// Represents the days of the week.
{attribute 'qualified_only'}
{attribute 'to_string'}
TYPE E_DayOfWeek :
(
	_ := 0, // Uninitialised or default value, representing an undefined day.
	Monday,
	Tuesday,
	Wednesday,
	Thursday,
	Friday,
	Saturday,
	Sunday
) UINT;
END_TYPE

(* stored: Version 1.1.0.1
   EnumerationTextList E_DayOfWeek: Id {bff4f9ca-233b-032b-1b58-0ffa422b15b2} *)
